PROGRAM MAIN
VAR
	
END_VAR

POU_Test();

END_PROGRAM

(* stored: Version 1.1.0.1, ProductVersion 3.1.4024.12
   POU MAIN: Id {ed1eb1bb-ebe0-40ad-a474-54e62c8f6397}, SpecialFunc None *)
